// TIA Portal V18 export
TYPE "LGasp_typeHMI_stazione"
// stored: IsFailsafeCompliant false
   STRUCT
      abilitata : Bool;   // Stazione abilitata
      invisibile : Bool;   // Invisibile sul sinottico, serve solo per visualizzazione allarmi
      zona : DInt;   // Indice array delle zone
      nome : WString[20];   // Nome della stazione
      nometrad : WString[20];   // Nome della stazione tradotto in lingua cliente
      AUTOman : Bool;   // 1=automatico 0=manuale
      MARCIAstop : Bool;   // 1=marcia 0=stop
      allarmi : Bool;   // Allami presente nella stazione
      warning : Bool;   // Warning presente nella stazione
      ds : Array[1.."N_DS"] of "LGasp_typeHMI_DS";   // Dati settings
      all { ExternalAccessible := 'False'; ExternalVisible := 'False'; ExternalWritable := 'False'} : Array[1..192] of Bool;   // Allarmi
      allarmipc : Array[1..6] of DInt;
      war { ExternalAccessible := 'False'; ExternalVisible := 'False'; ExternalWritable := 'False'} : Array[1..32] of Bool;   // Warning
      warningpc : DInt;
   END_STRUCT;
END_TYPE
